FUNCTION_BLOCK fis_cfc
VAR_INPUT
	crispinput1:real;
END_VAR

VAR
mymf:MEMBERSHIP_FUNCTION:=(mymf.Name:='error',Points:=[1,2,3,4,5]);
END_VAR

VAR_OUTPUT
END_VAR
VAR
	FB_FIS_0: fb_fis;
END_VAR
VAR // added by the converter: edge detectors and wires of the graphical bodies
    _w1, _w2, _w3 : BOOL;
END_VAR

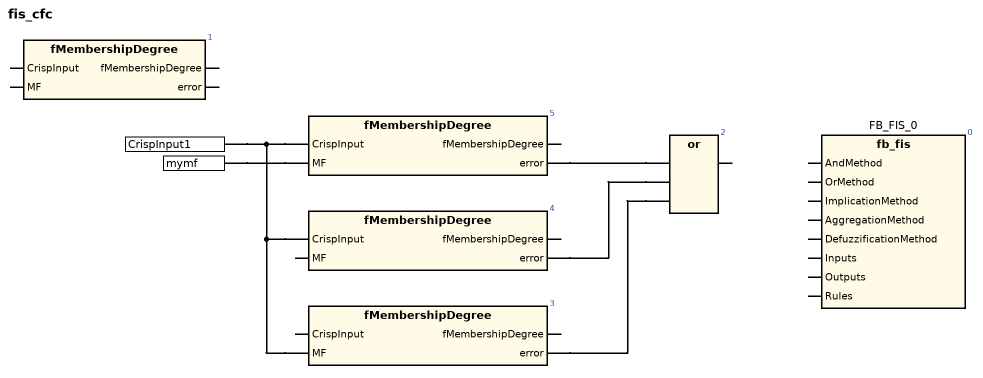
FB_FIS_0(); // fb_fis
fMembershipDegree();
(* _w1 OR _w2 OR _w3; result not used *)
fMembershipDegree(MF := CrispInput1, error => _w3);
fMembershipDegree(CrispInput := CrispInput1, error => _w2);
fMembershipDegree(CrispInput := CrispInput1, MF := mymf, error => _w1);

END_FUNCTION_BLOCK

(* stored: Version 1.1.0.1, ProductVersion 3.1.4024.6
   POU fis_cfc: Id {7483790b-fd8b-4a7d-bc62-44868d8ec0fb}, SpecialFunc None *)
